SUBAPPLICATION Uebung_002a6_AX2 (* DigitalInput_I1-3 mit AND auf DigitalOutput_Q1, mit Plug and Socket *)
  (* Standard: 61499-2; Description: Copyright (c) 2023 Meisterschulen am Ostbahnhof This program and the accompanying materials are made available under the terms of the Eclipse Public License 2.0 which is available at https://www.eclipse.org/legal/epl-2.0/ SPDX-License-Identifier: EPL-2.0 *)
  (* Version 1.0, 2023-10-23, Franz Höpfinger, Meisterschulen am Ostbahnhof *)
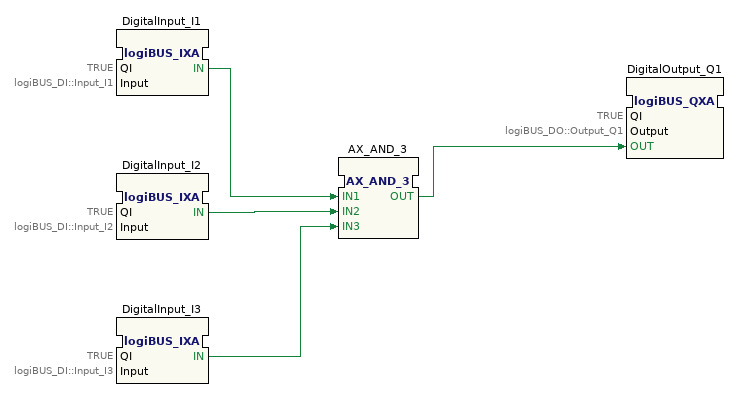
  FBS
    DigitalInput_I1 : logiBUS_IXA(QI := TRUE, Input := logiBUS_DI::Input_I1);
    DigitalOutput_Q1 : logiBUS_QXA(QI := TRUE, Output := logiBUS_DO::Output_Q1);
    AX_AND_3 : AX_AND_3;
    DigitalInput_I2 : logiBUS_IXA(QI := TRUE, Input := logiBUS_DI::Input_I2);
    DigitalInput_I3 : logiBUS_IXA(QI := TRUE, Input := logiBUS_DI::Input_I3);
  END_FBS
  ADAPTER_CONNECTIONS
    AX_AND_3.OUT TO DigitalOutput_Q1.OUT;
    DigitalInput_I1.IN TO AX_AND_3.IN1;
    DigitalInput_I2.IN TO AX_AND_3.IN2;
    DigitalInput_I3.IN TO AX_AND_3.IN3;
  END_CONNECTIONS
END_SUBAPPLICATION
